// TIA Portal V20 export
VAR_GLOBAL   // PLC tag table "HMI Tags"
   HMI_Popup AT %MW1104 : Word;
   HMI_ForwardJog_Button AT %I1.4 : Bool;
   HMI_BackwardJog_Button AT %I1.5 : Bool;
   HMI_Servo_Velocity_Conversion AT %MD1 : Real;
   HMI_Popup_Result AT %MW1106 : Word;
   HMI_Result AT %MW1108 : Word;
   HMI_Screen_Number AT %MW1100 : Word;
   HMI_Gate_Opener AT %M1.6 : Bool;
END_VAR
